(* IEC 61131-3 sources: Industry-PLC-LLM/data/PLCBEAD_repo/PLCBEAD_PLCEmbed-main/PLC-BEAD/Source/GEB/SHR1, 1 file *)

(* ---- SHR1.ST ---- *)
FUNCTION SHR1 :DWORD

	VAR_INPUT
		IN :	DWORD;
		N :	INT;
	END_VAR

	SHR1  := SHL(DWORD#16#FF_FF_FF_FF,32-N) OR SHR(IN,N);

END_FUNCTION

PROGRAM program0

	VAR
		IN : DWORD;
		N :	INT;
		CEIL5_OUT : DWORD;
	END_VAR

	CEIL5_OUT := SHR1 (IN, N);

END_PROGRAM
